# EPICS substitutions: apps/mpodLvApp/Db/htcc-iseg.substitutions
file "db/mpod-crate.db" {
pattern { HOST }
        { hvhtcc1 }
}

file "db/iseg-module.db" {
pattern { HOST HOSTNAME MX }
        { 129.57.161.15 hvhtcc1 1 }
        { 129.57.161.15 hvhtcc1 2 }
        { 129.57.161.15 hvhtcc1 3 }
        { 129.57.161.15 hvhtcc1 4 }
}

file "db/iseg-channel.db" {
pattern { HVHOST HV HVCH }
        { 129.57.161.15 B_DET_HTCC_HV_SEC1_L1 1 }
        { 129.57.161.15 B_DET_HTCC_HV_SEC1_L2 2 }
        { 129.57.161.15 B_DET_HTCC_HV_SEC1_L3 3 }
        { 129.57.161.15 B_DET_HTCC_HV_SEC1_L4 4 }
        { 129.57.161.15 B_DET_HTCC_HV_SEC1_R1 5 }
        { 129.57.161.15 B_DET_HTCC_HV_SEC1_R2 6 }
        { 129.57.161.15 B_DET_HTCC_HV_SEC1_R3 7 }
        { 129.57.161.15 B_DET_HTCC_HV_SEC1_R4 8 }
        { 129.57.161.15 B_DET_HTCC_HV_SEC2_L1 9 }
        { 129.57.161.15 B_DET_HTCC_HV_SEC2_L2 10 }
        { 129.57.161.15 B_DET_HTCC_HV_SEC2_L3 11 }
        { 129.57.161.15 B_DET_HTCC_HV_SEC2_L4 12 }
        { 129.57.161.15 B_DET_HTCC_HV_SEC2_R1 13 }
        { 129.57.161.15 B_DET_HTCC_HV_SEC2_R2 14 }
        { 129.57.161.15 B_DET_HTCC_HV_SEC2_R3 15 }
        { 129.57.161.15 B_DET_HTCC_HV_SEC2_R4 16 }
        { 129.57.161.15 B_DET_HTCC_HV_SEC3_L1 101 }
        { 129.57.161.15 B_DET_HTCC_HV_SEC3_L2 102 }
        { 129.57.161.15 B_DET_HTCC_HV_SEC3_L3 103 }
        { 129.57.161.15 B_DET_HTCC_HV_SEC3_L4 104 }
        { 129.57.161.15 B_DET_HTCC_HV_SEC3_R1 105 }
        { 129.57.161.15 B_DET_HTCC_HV_SEC3_R2 106 }
        { 129.57.161.15 B_DET_HTCC_HV_SEC3_R3 107 }
        { 129.57.161.15 B_DET_HTCC_HV_SEC3_R4 108 }
        { 129.57.161.15 B_DET_HTCC_HV_SEC4_L1 109 }
        { 129.57.161.15 B_DET_HTCC_HV_SEC4_L2 110 }
        { 129.57.161.15 B_DET_HTCC_HV_SEC4_L3 111 }
        { 129.57.161.15 B_DET_HTCC_HV_SEC4_L4 112 }
        { 129.57.161.15 B_DET_HTCC_HV_SEC4_R1 113 }
        { 129.57.161.15 B_DET_HTCC_HV_SEC4_R2 114 }
        { 129.57.161.15 B_DET_HTCC_HV_SEC4_R3 115 }
        { 129.57.161.15 B_DET_HTCC_HV_SEC4_R4 116 }
        { 129.57.161.15 B_DET_HTCC_HV_SEC5_L1 201 }
        { 129.57.161.15 B_DET_HTCC_HV_SEC5_L2 202 }
        { 129.57.161.15 B_DET_HTCC_HV_SEC5_L3 203 }
        { 129.57.161.15 B_DET_HTCC_HV_SEC5_L4 204 }
        { 129.57.161.15 B_DET_HTCC_HV_SEC5_R1 205 }
        { 129.57.161.15 B_DET_HTCC_HV_SEC5_R2 206 }
        { 129.57.161.15 B_DET_HTCC_HV_SEC5_R3 207 }
        { 129.57.161.15 B_DET_HTCC_HV_SEC5_R4 208 }
        { 129.57.161.15 B_DET_HTCC_HV_SEC6_L1 209 }
        { 129.57.161.15 B_DET_HTCC_HV_SEC6_L2 210 }
        { 129.57.161.15 B_DET_HTCC_HV_SEC6_L3 211 }
        { 129.57.161.15 B_DET_HTCC_HV_SEC6_L4 212 }
        { 129.57.161.15 B_DET_HTCC_HV_SEC6_R1 213 }
        { 129.57.161.15 B_DET_HTCC_HV_SEC6_R2 214 }
        { 129.57.161.15 B_DET_HTCC_HV_SEC6_R3 215 }
        { 129.57.161.15 B_DET_HTCC_HV_SEC6_R4 216 }
}
